(* IEC 61131-3 sources: AXOpen/src/integrations/app/src/IntegrationTests/data, 2 files *)

(* ---- AxoDataFragmentExchange.st ---- *)
USING AXOpen.Core;
USING AXOpen.Data;
USING AXOpen.Probers;

NAMESPACE IntegrationAxoDataFramentsExchange

    {S7.extern=ReadWrite}
    CLASS AxoDataFragmentExchangeContext EXTENDS AXOpen.Core.AxoContext
        VAR PUBLIC
            PD : ProcessData;
            CreateTest : DataCreateTest;
            ReadTest : DataReadTest;
            UpdateTest : DataUpdateTest;
            DeleteTest : DataDeleteTest;
            _rootObject :   AxoObject;
        END_VAR

        METHOD PROTECTED OVERRIDE Main
            _rootObject.InitializeWithContext(THIS);

            PD.Run(_rootObject);

            CreateTest.InjectManger(PD);
            CreateTest.Run(_rootObject);

            ReadTest.InjectManger(PD);
            ReadTest.Run(_rootObject);

            DeleteTest.InjectManger(PD);
            DeleteTest.Run(_rootObject);

            UpdateTest.InjectManger(PD);
            UpdateTest.Run(_rootObject);
        END_METHOD

    END_CLASS

    {S7.extern=ReadWrite}
    CLASS ProcessData EXTENDS AXOpen.Data.AxoDataFragmentExchange
        VAR PUBLIC
            {#ix-attr:[AXOpen.Data.AxoDataFragmentAttribute]}
            Set : SharedProductionDataManager;
            {#ix-attr:[AXOpen.Data.AxoDataFragmentAttribute]}
            Manip : FragmentProcessDataManger;
        END_VAR
    END_CLASS

    {S7.extern=ReadWrite}
    CLASS SharedProductionData EXTENDS AXOpen.Data.AxoDataEntity
        VAR PUBLIC
            ComesFrom : INT;
            GoesTo : INT;
        END_VAR
    END_CLASS

    {S7.extern=ReadWrite}
    CLASS SharedProductionDataManager EXTENDS AXOpen.Data.AxoDataExchange
        VAR PUBLIC
            {#ix-generic:TOnline}
            {#ix-generic:TPlain as POCO}
            {#ix-attr:[AXOpen.Data.AxoDataEntityAttribute]}
            {#ix-attr:[Container(Layout.Stack)]}
            Set : SharedProductionData;
        END_VAR
    END_CLASS

    {S7.extern=ReadWrite}
    CLASS FragmentProcessDataManger
        EXTENDS AXOpen.Data.AxoDataExchange
        VAR PUBLIC
            {#ix-generic:TOnline}
            {#ix-generic:TPlain as POCO}
            {#ix-attr:[AXOpen.Data.AxoDataEntityAttribute]}
            {#ix-attr:[Container(Layout.Stack)]}
            Set : FragmentProcessData;
        END_VAR
    END_CLASS

    {S7.extern=ReadWrite}
    CLASS FragmentProcessData
        EXTENDS AXOpen.Data.AxoDataEntity
        VAR PUBLIC
            CounterDelay : ULINT;
        END_VAR
    END_CLASS

    {S7.extern=ReadWrite}
    CLASS DataCreateTest EXTENDS AxoProberWithCompletedCondition
        VAR PUBLIC
            Manager : IAxoDataExchange;
            Identifier : STRING[254];
        END_VAR
        METHOD PROTECTED OVERRIDE Test : BOOL
            VAR
                _taskState : IAxoTaskState;
            END_VAR
            IF(Manager <> NULL) THEN
                _taskState := Manager.Create(Identifier);
                THIS.ThrowWhen(_taskState.HasError(), _taskState.GetErrorDetails());
                Test := _taskState.IsDone();
            END_IF;
        END_METHOD

        METHOD OVERRIDE OnRestore
            SUPER.OnRestore();
            IF(Manager <> NULL) THEN
                 Manager.Restore();
            END_IF;
        END_METHOD

        METHOD PUBLIC InjectManger
            VAR_INPUT
                Injectee : IAxoDataExchange;
            END_VAR
            Manager := Injectee;
        END_METHOD
    END_CLASS

    {S7.extern=ReadWrite}
    CLASS DataReadTest EXTENDS AxoProberWithCompletedCondition
        VAR PUBLIC
            Manager : IAxoDataExchange;
            Identifier : STRING[254];
        END_VAR
        METHOD PROTECTED OVERRIDE Test : BOOL
            VAR
                _taskState : IAxoTaskState;
            END_VAR
            IF(Manager <> NULL) THEN
                _taskState := Manager.Read(Identifier);
                THIS.ThrowWhen(_taskState.HasError(), _taskState.GetErrorDetails());
                Test := _taskState.IsDone();
            END_IF;
        END_METHOD

        METHOD OVERRIDE OnRestore
            SUPER.OnRestore();
            IF(Manager <> NULL) THEN
                 Manager.Restore();
            END_IF;
        END_METHOD

        METHOD PUBLIC InjectManger
            VAR_INPUT
                Injectee : IAxoDataExchange;
            END_VAR
            Manager := Injectee;
        END_METHOD
    END_CLASS

    {S7.extern=ReadWrite}
    CLASS DataUpdateTest EXTENDS AxoProberWithCompletedCondition
        VAR PUBLIC
            Manager : IAxoDataExchange;
            Identifier : STRING[254];
        END_VAR
        METHOD PROTECTED OVERRIDE Test : BOOL
            VAR
                _taskState : IAxoTaskState;
            END_VAR
            IF(Manager <> NULL) THEN
                _taskState := Manager.Update(Identifier);
                THIS.ThrowWhen(_taskState.HasError(), _taskState.GetErrorDetails());
                Test := _taskState.IsDone();
            END_IF;
        END_METHOD

        METHOD OVERRIDE OnRestore
            SUPER.OnRestore();
            IF(Manager <> NULL) THEN
                 Manager.Restore();
            END_IF;
        END_METHOD

        METHOD PUBLIC InjectManger
            VAR_INPUT
                Injectee : IAxoDataExchange;
            END_VAR
            Manager := Injectee;
        END_METHOD
    END_CLASS

    {S7.extern=ReadWrite}
    CLASS DataDeleteTest EXTENDS AxoProberWithCompletedCondition
        VAR PUBLIC
            Manager : IAxoDataExchange;
            Identifier : STRING[254];
        END_VAR
        METHOD PROTECTED OVERRIDE Test : BOOL
            VAR
                _taskState : IAxoTaskState;
            END_VAR
            IF(Manager <> NULL) THEN
                _taskState := Manager.Delete(Identifier);
                THIS.ThrowWhen(_taskState.HasError(), _taskState.GetErrorDetails());
                Test := _taskState.IsDone();
            END_IF;
        END_METHOD

        METHOD OVERRIDE OnRestore
            SUPER.OnRestore();
            IF(Manager <> NULL) THEN
                 Manager.Restore();
            END_IF;
        END_METHOD

        METHOD PUBLIC InjectManger
            VAR_INPUT
                Injectee : IAxoDataExchange;
            END_VAR
            Manager := Injectee;
        END_METHOD
    END_CLASS
END_NAMESPACE

(* ---- DataExchangeLightTests.st ---- *)
USING AXOpen.Core;
USING AXOpen.Data;
USING AXOpen.Probers;

NAMESPACE IntegrationLightDirect
    {S7.extern=ReadWrite}
    CLASS DataExchangeLightTestsContext EXTENDS AxoContext
        VAR PUBLIC
            DM : IAxoDataExchange;
            CreateTest : DataCreateTest;
            ReadTest : DataReadTest;
            UpdateTest : DataUpdateTest;
            DeleteTest : DataDeleteTest;
            _rootObject : AxoObject;
        END_VAR

        METHOD PUBLIC InjectDM
            VAR_INPUT
                iDM : IAxoDataExchange;
            END_VAR
            DM := iDM;
        END_METHOD

        METHOD PROTECTED OVERRIDE Main
            THIS.InitializeRootObject(_rootObject);
            CreateTest.InjectManger(DM);
            CreateTest.Run(_rootObject);

            ReadTest.InjectManger(DM);
            ReadTest.Run(_rootObject);

            DeleteTest.InjectManger(DM);
            DeleteTest.Run(_rootObject);

            UpdateTest.InjectManger(DM);
            UpdateTest.Run(_rootObject);

        END_METHOD
    END_CLASS

    {S7.extern=ReadWrite}
    CLASS DataCreateTest EXTENDS AxoProberWithCompletedCondition
        VAR PUBLIC
            Manager : IAxoDataExchange;
            Identifier : STRING[254];
        END_VAR
        METHOD PROTECTED OVERRIDE Test : BOOL
            VAR
                _taskState : IAxoTaskState;
            END_VAR
            IF(Manager <> NULL) THEN
                _taskState := Manager.Create(Identifier);
                THIS.ThrowWhen(_taskState.HasError(), _taskState.GetErrorDetails());
                Test := _taskState.IsDone();
            END_IF;
        END_METHOD

        METHOD OVERRIDE OnRestore
            SUPER.OnRestore();
            IF(Manager <> NULL) THEN
                 Manager.Restore();
            END_IF;
        END_METHOD

        METHOD PUBLIC InjectManger
            VAR_INPUT
                Injectee : IAxoDataExchange;
            END_VAR
            Manager := Injectee;
        END_METHOD
    END_CLASS

    {S7.extern=ReadWrite}
    CLASS DataReadTest EXTENDS AxoProberWithCompletedCondition
        VAR PUBLIC
            Manager : IAxoDataExchange;
            Identifier : STRING[254];
        END_VAR
        METHOD PROTECTED OVERRIDE Test : BOOL
            VAR
                _taskState : IAxoTaskState;
            END_VAR
            IF(Manager <> NULL) THEN
                _taskState := Manager.Read(Identifier);
                THIS.ThrowWhen(_taskState.HasError(), _taskState.GetErrorDetails());
                Test := _taskState.IsDone();
            END_IF;
        END_METHOD

        METHOD OVERRIDE OnRestore
            SUPER.OnRestore();
            IF(Manager <> NULL) THEN
                 Manager.Restore();
            END_IF;
        END_METHOD

        METHOD PUBLIC InjectManger
            VAR_INPUT
                Injectee : IAxoDataExchange;
            END_VAR
            Manager := Injectee;
        END_METHOD
    END_CLASS

    {S7.extern=ReadWrite}
    CLASS DataUpdateTest EXTENDS AxoProberWithCompletedCondition
        VAR PUBLIC
            Manager : IAxoDataExchange;
            Identifier : STRING[254];
        END_VAR
        METHOD PROTECTED OVERRIDE Test : BOOL
            VAR
                _taskState : IAxoTaskState;
            END_VAR
            IF(Manager <> NULL) THEN
                _taskState := Manager.Update(Identifier);
                THIS.ThrowWhen(_taskState.HasError(), _taskState.GetErrorDetails());
                Test := _taskState.IsDone();
            END_IF;
        END_METHOD

        METHOD OVERRIDE OnRestore
            SUPER.OnRestore();
            IF(Manager <> NULL) THEN
                 Manager.Restore();
            END_IF;
        END_METHOD

        METHOD PUBLIC InjectManger
            VAR_INPUT
                Injectee : IAxoDataExchange;
            END_VAR
            Manager := Injectee;
        END_METHOD
    END_CLASS

    {S7.extern=ReadWrite}
    CLASS DataDeleteTest EXTENDS AxoProberWithCompletedCondition
        VAR PUBLIC
            Manager : IAxoDataExchange;
            Identifier : STRING[254];
        END_VAR
        METHOD PROTECTED OVERRIDE Test : BOOL
            VAR
                _taskState : IAxoTaskState;
            END_VAR
            IF(Manager <> NULL) THEN
                _taskState := Manager.Delete(Identifier);
                THIS.ThrowWhen(_taskState.HasError(), _taskState.GetErrorDetails());
                Test := _taskState.IsDone();
            END_IF;
        END_METHOD

        METHOD OVERRIDE OnRestore
            SUPER.OnRestore();
            IF(Manager <> NULL) THEN
                 Manager.Restore();
            END_IF;
        END_METHOD

        METHOD PUBLIC InjectManger
            VAR_INPUT
                Injectee : IAxoDataExchange;
            END_VAR
            Manager := Injectee;
        END_METHOD
    END_CLASS

    {S7.extern=ReadWrite}
    CLASS DataManager EXTENDS AXOpen.Data.AxoDataExchange
        VAR PUBLIC
            {#ix-generic:TOnline}
            {#ix-generic:TPlain as POCO}
            {#ix-attr:[AxoDataEntityAttribute]}
            _data       : DataSet;
        END_VAR
    END_CLASS

    {S7.extern=ReadWrite}
    CLASS DataSet EXTENDS AXOpen.Data.AxoDataEntity
        VAR PUBLIC
            SomeData : STRING;
        END_VAR
    END_CLASS

END_NAMESPACE
